Omron CX-Programmer project 新工程 (CX-Programmer 9.73)

# PLC 新PLC1: CQM1H CPU21

## Program 新程序1 (no task)
; 上传一个欧姆龙程序，轴承数控磨床用的。该程序控制三台步进电机。 / 系统涉及的物理设备包括操作面板按钮、传感器、砂轮电机、进给电机和冷却泵。 / 系统通过自动模式启动按钮启动整个流程，操作员按下后，工件在进给电机控制信号驱动下被送入加工位置，由工件位置传感器1确认到位后，砂轮电机控制信号激活砂轮开始磨削。 / 为确保加工质量，加工进行中标志置位时，冷却泵启动信号必须保持激活，提供持续的冷却液，防止工件过热损坏。 / 在加工进行中标志激活时，通过定时器确保冷却泵启动信号持续运行。 / 当工件位置传感器1确认工件到位后，砂轮电机控制信号才会被激活，避免空转浪费能源或损伤设备。 / 在手动模式下，进给电机启动按钮置位控制信号，进而驱动进给电机。 / 在自动模式启动按钮置位时，进给电机控制信号不会被手动触发。 / 进给过程中，进给脉冲信号根据数据存储区1设置的脉冲数精确控制步进电机，确保工件定位无偏差。 / 加工完成后，退料启用标志置位时，系统触发退料步骤将工件退出，避免工件滞留造成设备堵塞。 / 当退料启用标志置位时，若系统处于自动流程，触发退料步骤。 / 当工件位置传感器2检测工件离开时，流程结束并记录状态至数据存储区2。

### Section 段1

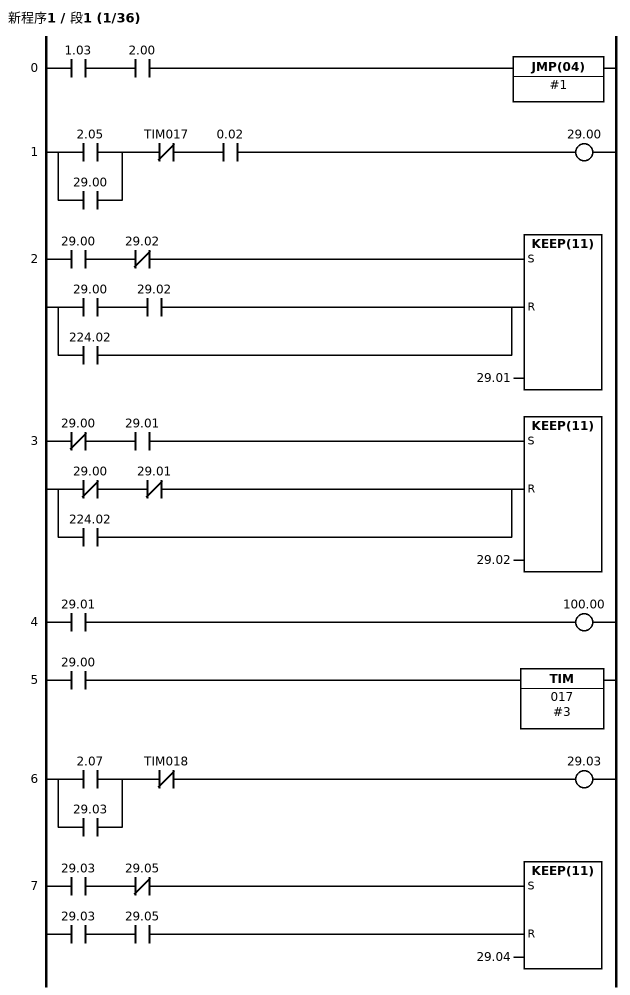
; rung 0
LD 1.03
AND 2.00
JMP(04) #1
; rung 1
LD 2.05
OR 29.00
ANDNOT TIM017
AND 0.02
OUT 29.00
; rung 2
LD 29.00
ANDNOT 29.02
LD 29.00
AND 29.02
OR 224.02
KEEP(11) 29.01
; rung 3
LDNOT 29.00
AND 29.01
LDNOT 29.00
ANDNOT 29.01
OR 224.02
KEEP(11) 29.02
; rung 4
LD 29.01
OUT 100.00
; rung 5
LD 29.00
TIM 017 #3
; rung 6
LD 2.07
OR 29.03
ANDNOT TIM018
OUT 29.03
; rung 7
LD 29.03
ANDNOT 29.05
LD 29.03
AND 29.05
KEEP(11) 29.04

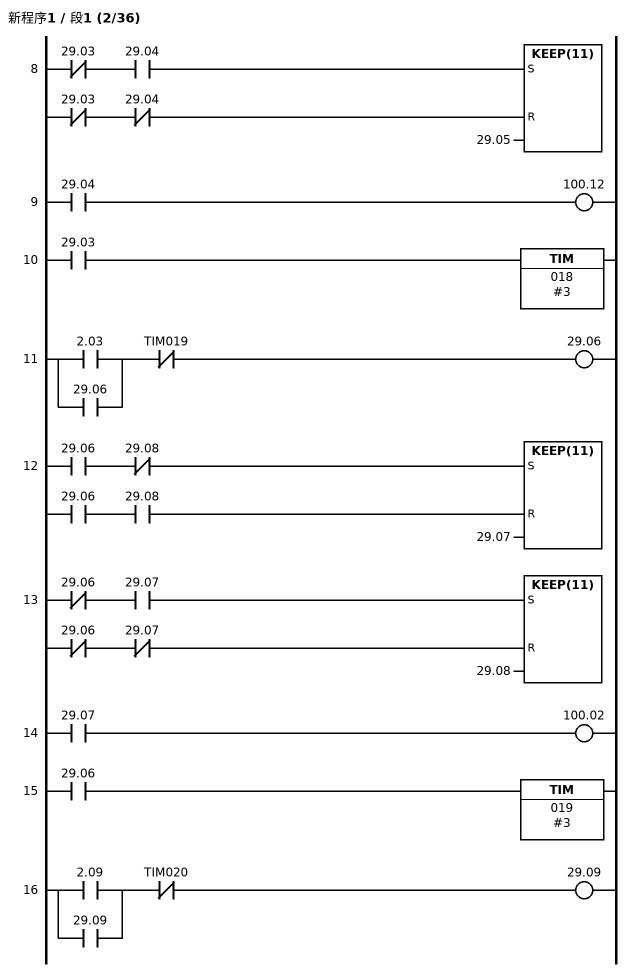
; rung 8
LDNOT 29.03
AND 29.04
LDNOT 29.03
ANDNOT 29.04
KEEP(11) 29.05
; rung 9
LD 29.04
OUT 100.12
; rung 10
LD 29.03
TIM 018 #3
; rung 11
LD 2.03
OR 29.06
ANDNOT TIM019
OUT 29.06
; rung 12
LD 29.06
ANDNOT 29.08
LD 29.06
AND 29.08
KEEP(11) 29.07
; rung 13
LDNOT 29.06
AND 29.07
LDNOT 29.06
ANDNOT 29.07
KEEP(11) 29.08
; rung 14
LD 29.07
OUT 100.02
; rung 15
LD 29.06
TIM 019 #3
; rung 16
LD 2.09
OR 29.09
ANDNOT TIM020
OUT 29.09

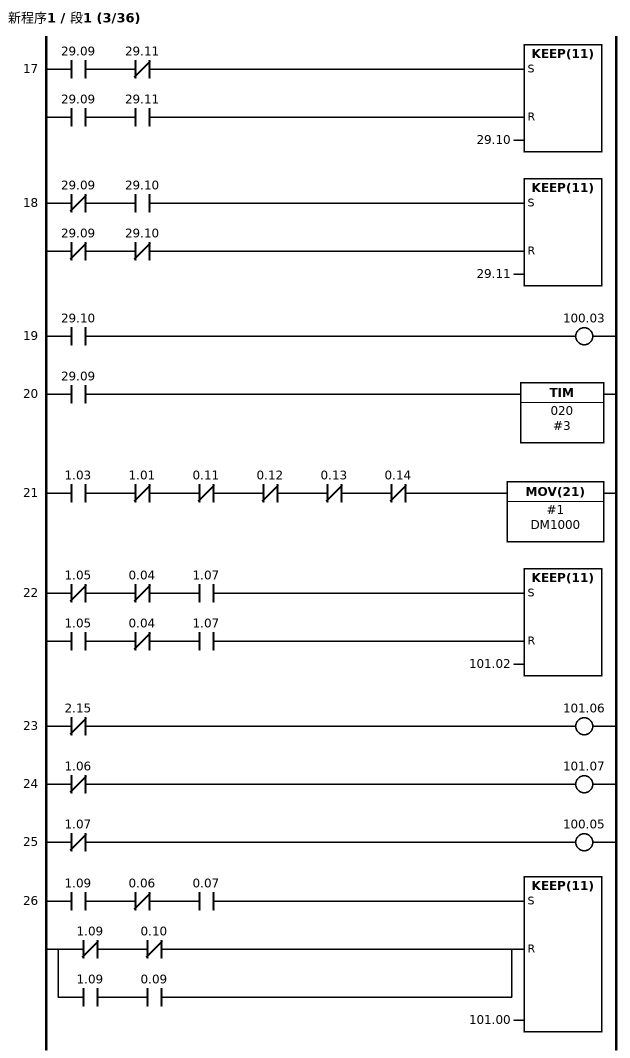
; rung 17
LD 29.09
ANDNOT 29.11
LD 29.09
AND 29.11
KEEP(11) 29.10
; rung 18
LDNOT 29.09
AND 29.10
LDNOT 29.09
ANDNOT 29.10
KEEP(11) 29.11
; rung 19
LD 29.10
OUT 100.03
; rung 20
LD 29.09
TIM 020 #3
; rung 21
LD 1.03
ANDNOT 1.01
ANDNOT 0.11
ANDNOT 0.12
ANDNOT 0.13
ANDNOT 0.14
MOV(21) #1 DM1000
; rung 22
LDNOT 1.05
ANDNOT 0.04
AND 1.07
LD 1.05
ANDNOT 0.04
AND 1.07
KEEP(11) 101.02
; rung 23
LDNOT 2.15
OUT 101.06
; rung 24
LDNOT 1.06
OUT 101.07
; rung 25
LDNOT 1.07
OUT 100.05
; rung 26
LD 1.09
ANDNOT 0.06
AND 0.07
LDNOT 1.09
ANDNOT 0.10
LD 1.09
AND 0.09
ORLD
KEEP(11) 101.00

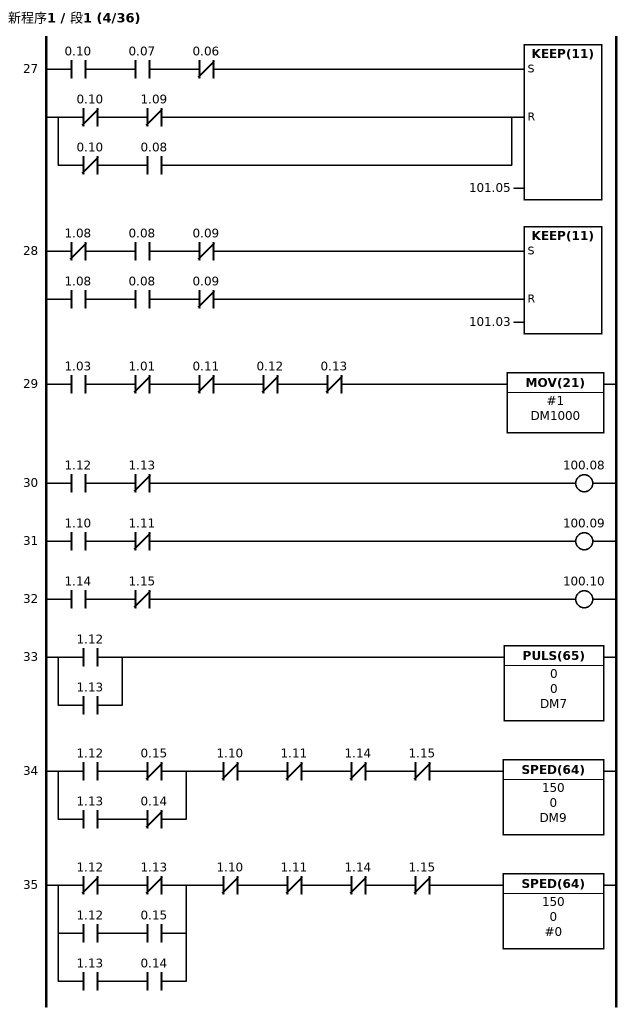
; rung 27
LD 0.10
AND 0.07
ANDNOT 0.06
LDNOT 0.10
ANDNOT 1.09
LDNOT 0.10
AND 0.08
ORLD
KEEP(11) 101.05
; rung 28
LDNOT 1.08
AND 0.08
ANDNOT 0.09
LD 1.08
AND 0.08
ANDNOT 0.09
KEEP(11) 101.03
; rung 29
LD 1.03
ANDNOT 1.01
ANDNOT 0.11
ANDNOT 0.12
ANDNOT 0.13
MOV(21) #1 DM1000
; rung 30
LD 1.12
ANDNOT 1.13
OUT 100.08
; rung 31
LD 1.10
ANDNOT 1.11
OUT 100.09
; rung 32
LD 1.14
ANDNOT 1.15
OUT 100.10
; rung 33
LD 1.12
OR 1.13
PULS(65) 0 0 DM7
; rung 34
LD 1.12
ANDNOT 0.15
LD 1.13
ANDNOT 0.14
ORLD
ANDNOT 1.10
ANDNOT 1.11
ANDNOT 1.14
ANDNOT 1.15
SPED(64) 150 0 DM9
; rung 35
LDNOT 1.12
ANDNOT 1.13
LD 1.12
AND 0.15
ORLD
LD 1.13
AND 0.14
ORLD
ANDNOT 1.10
ANDNOT 1.11
ANDNOT 1.14
ANDNOT 1.15
SPED(64) 150 0 #0

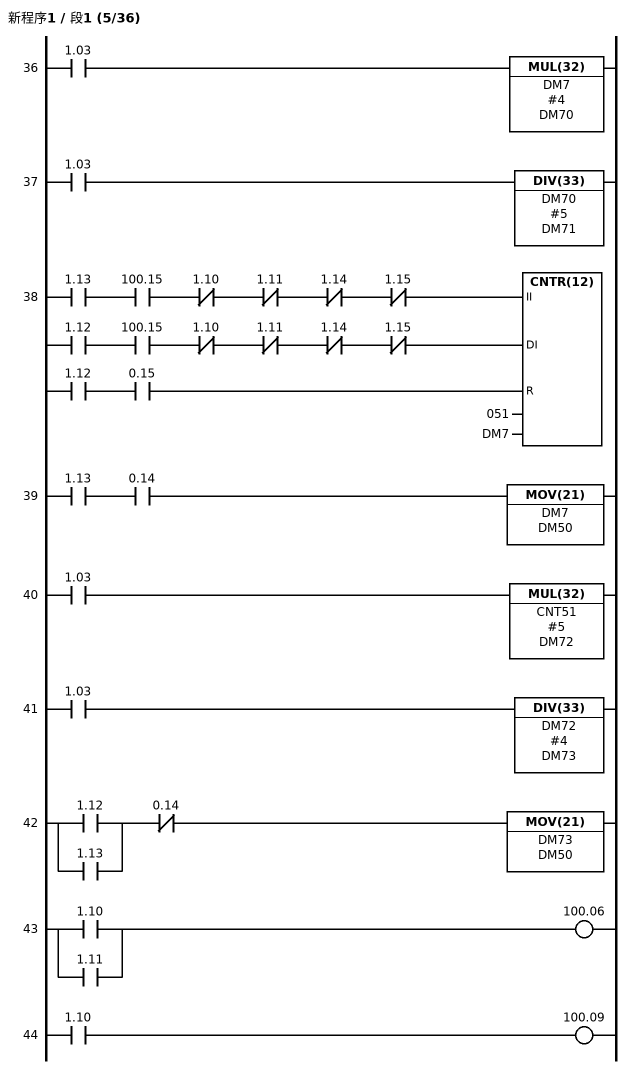
; rung 36
LD 1.03
MUL(32) DM7 #4 DM70
; rung 37
LD 1.03
DIV(33) DM70 #5 DM71
; rung 38
LD 1.13
AND 100.15
ANDNOT 1.10
ANDNOT 1.11
ANDNOT 1.14
ANDNOT 1.15
LD 1.12
AND 100.15
ANDNOT 1.10
ANDNOT 1.11
ANDNOT 1.14
ANDNOT 1.15
LD 1.12
AND 0.15
CNTR(12) 051 DM7
; rung 39
LD 1.13
AND 0.14
MOV(21) DM7 DM50
; rung 40
LD 1.03
MUL(32) CNT51 #5 DM72
; rung 41
LD 1.03
DIV(33) DM72 #4 DM73
; rung 42
LD 1.12
OR 1.13
ANDNOT 0.14
MOV(21) DM73 DM50
; rung 43
LD 1.10
OR 1.11
OUT 100.06
; rung 44
LD 1.10
OUT 100.09

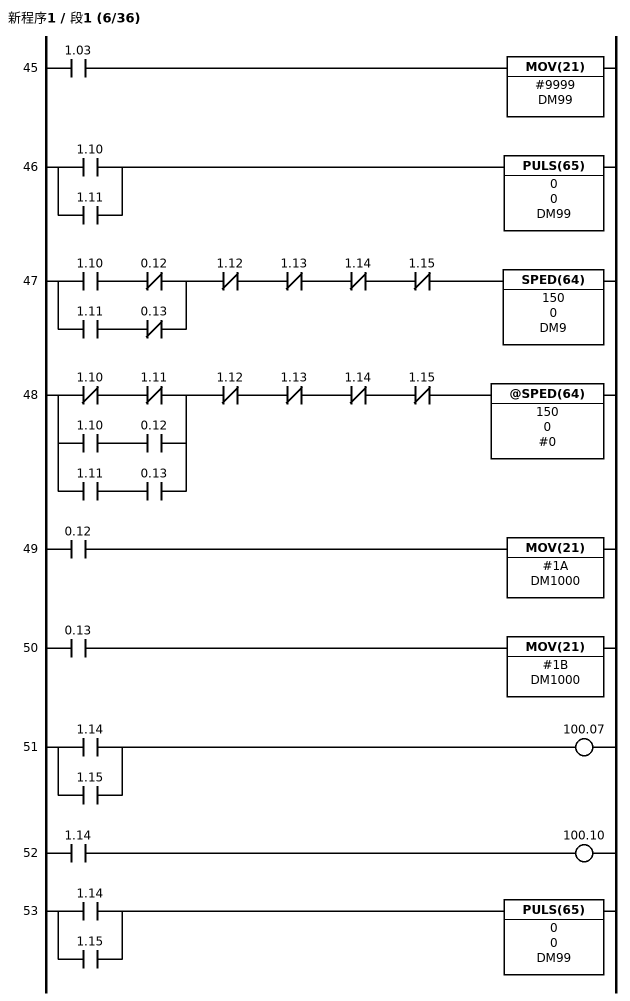
; rung 45
LD 1.03
MOV(21) #9999 DM99
; rung 46
LD 1.10
OR 1.11
PULS(65) 0 0 DM99
; rung 47
LD 1.10
ANDNOT 0.12
LD 1.11
ANDNOT 0.13
ORLD
ANDNOT 1.12
ANDNOT 1.13
ANDNOT 1.14
ANDNOT 1.15
SPED(64) 150 0 DM9
; rung 48
LDNOT 1.10
ANDNOT 1.11
LD 1.10
AND 0.12
ORLD
LD 1.11
AND 0.13
ORLD
ANDNOT 1.12
ANDNOT 1.13
ANDNOT 1.14
ANDNOT 1.15
@SPED(64) 150 0 #0
; rung 49
LD 0.12
MOV(21) #1A DM1000
; rung 50
LD 0.13
MOV(21) #1B DM1000
; rung 51
LD 1.14
OR 1.15
OUT 100.07
; rung 52
LD 1.14
OUT 100.10
; rung 53
LD 1.14
OR 1.15
PULS(65) 0 0 DM99

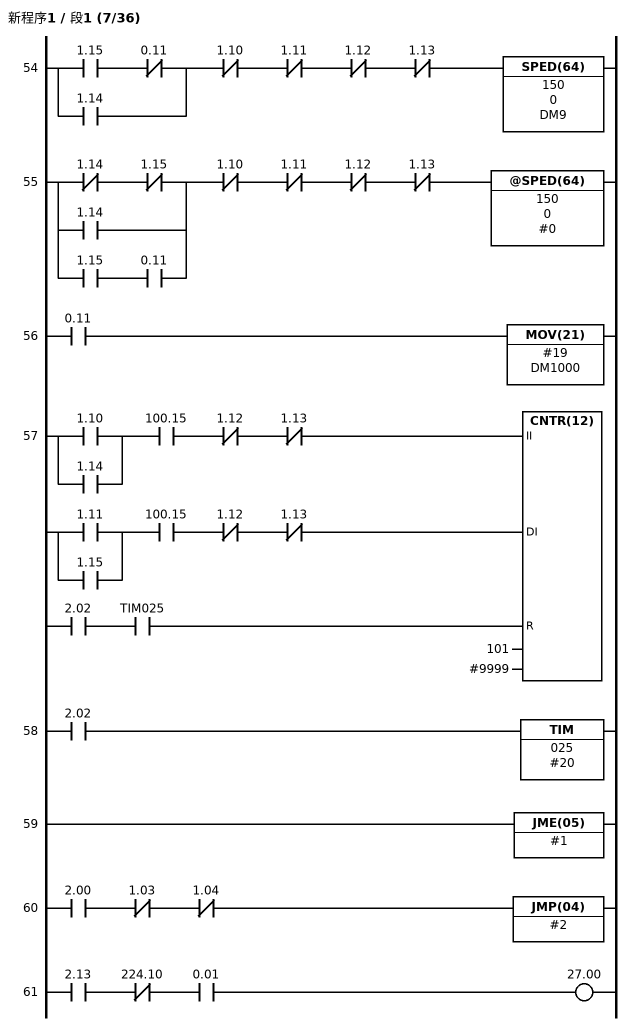
; rung 54
LD 1.15
ANDNOT 0.11
OR 1.14
ANDNOT 1.10
ANDNOT 1.11
ANDNOT 1.12
ANDNOT 1.13
SPED(64) 150 0 DM9
; rung 55
LDNOT 1.14
ANDNOT 1.15
OR 1.14
LD 1.15
AND 0.11
ORLD
ANDNOT 1.10
ANDNOT 1.11
ANDNOT 1.12
ANDNOT 1.13
@SPED(64) 150 0 #0
; rung 56
LD 0.11
MOV(21) #19 DM1000
; rung 57
LD 1.10
OR 1.14
AND 100.15
ANDNOT 1.12
ANDNOT 1.13
LD 1.11
OR 1.15
AND 100.15
ANDNOT 1.12
ANDNOT 1.13
LD 2.02
AND TIM025
CNTR(12) 101 #9999
; rung 58
LD 2.02
TIM 025 #20
; rung 59
JME(05) #1
; rung 60
LD 2.00
ANDNOT 1.03
ANDNOT 1.04
JMP(04) #2
; rung 61
LD 2.13
ANDNOT 224.10
AND 0.01
OUT 27.00

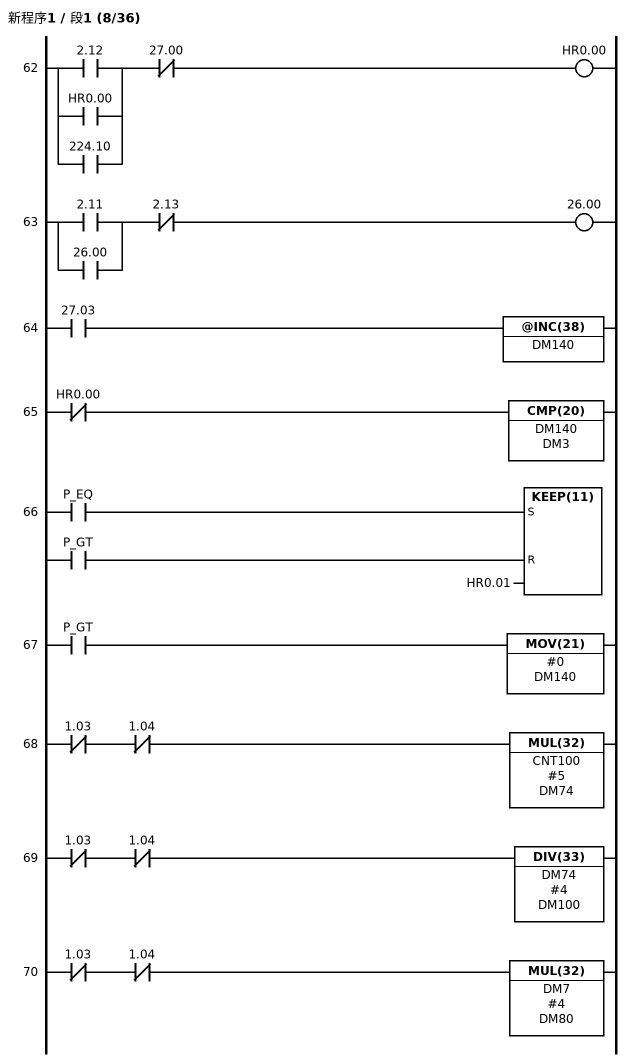
; rung 62
LD 2.12
OR HR0.00
OR 224.10
ANDNOT 27.00
OUT HR0.00
; rung 63
LD 2.11
OR 26.00
ANDNOT 2.13
OUT 26.00
; rung 64
LD 27.03
@INC(38) DM140
; rung 65
LDNOT HR0.00
CMP(20) DM140 DM3
; rung 66
LD P_EQ
LD P_GT
KEEP(11) HR0.01
; rung 67
LD P_GT
MOV(21) #0 DM140
; rung 68
LDNOT 1.03
ANDNOT 1.04
MUL(32) CNT100 #5 DM74
; rung 69
LDNOT 1.03
ANDNOT 1.04
DIV(33) DM74 #4 DM100
; rung 70
LDNOT 1.03
ANDNOT 1.04
MUL(32) DM7 #4 DM80

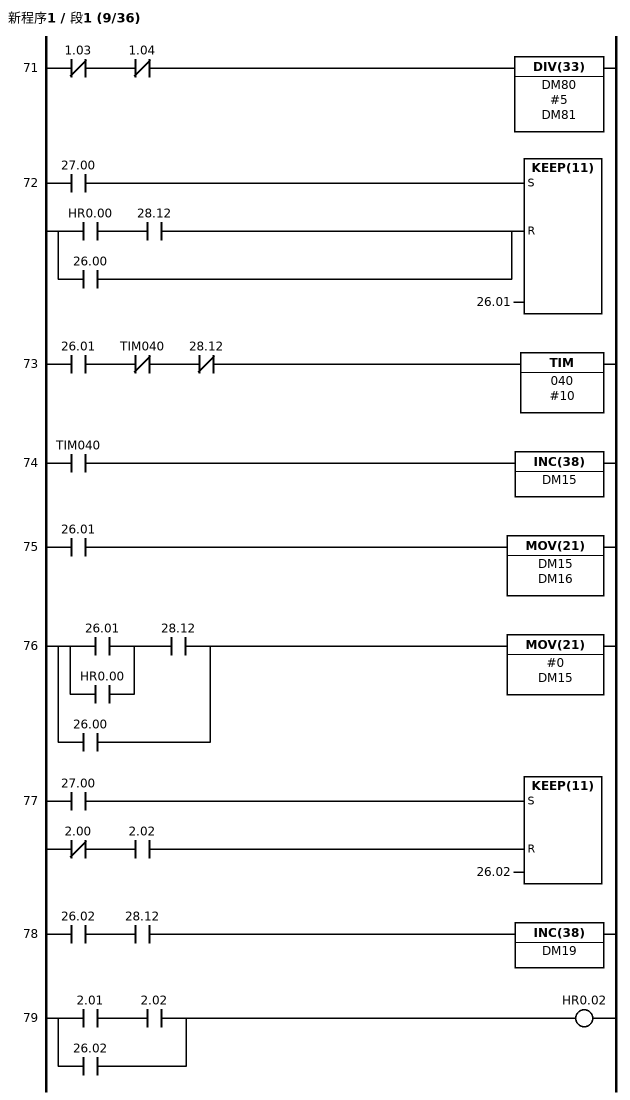
; rung 71
LDNOT 1.03
ANDNOT 1.04
DIV(33) DM80 #5 DM81
; rung 72
LD 27.00
LD HR0.00
AND 28.12
OR 26.00
KEEP(11) 26.01
; rung 73
LD 26.01
ANDNOT TIM040
ANDNOT 28.12
TIM 040 #10
; rung 74
LD TIM040
INC(38) DM15
; rung 75
LD 26.01
MOV(21) DM15 DM16
; rung 76
LD 26.01
OR HR0.00
AND 28.12
OR 26.00
MOV(21) #0 DM15
; rung 77
LD 27.00
LDNOT 2.00
AND 2.02
KEEP(11) 26.02
; rung 78
LD 26.02
AND 28.12
INC(38) DM19
; rung 79
LD 2.01
AND 2.02
OR 26.02
OUT HR0.02

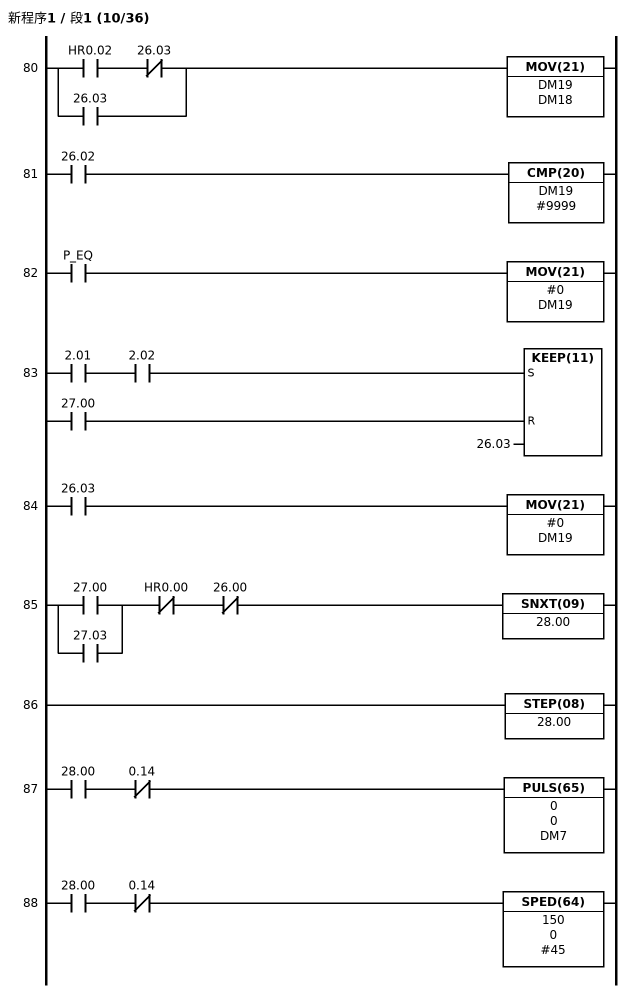
; rung 80
LD HR0.02
ANDNOT 26.03
OR 26.03
MOV(21) DM19 DM18
; rung 81
LD 26.02
CMP(20) DM19 #9999
; rung 82
LD P_EQ
MOV(21) #0 DM19
; rung 83
LD 2.01
AND 2.02
LD 27.00
KEEP(11) 26.03
; rung 84
LD 26.03
MOV(21) #0 DM19
; rung 85
LD 27.00
OR 27.03
ANDNOT HR0.00
ANDNOT 26.00
SNXT(09) 28.00
; rung 86
STEP(08) 28.00
; rung 87
LD 28.00
ANDNOT 0.14
PULS(65) 0 0 DM7
; rung 88
LD 28.00
ANDNOT 0.14
SPED(64) 150 0 #45

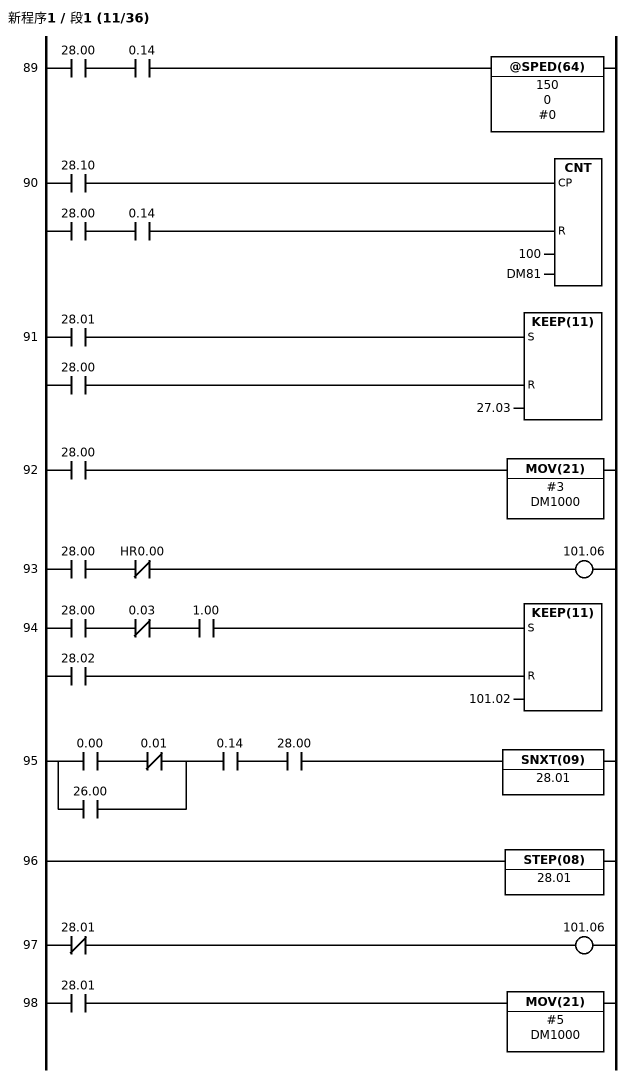
; rung 89
LD 28.00
AND 0.14
@SPED(64) 150 0 #0
; rung 90
LD 28.10
LD 28.00
AND 0.14
CNT 100 DM81
; rung 91
LD 28.01
LD 28.00
KEEP(11) 27.03
; rung 92
LD 28.00
MOV(21) #3 DM1000
; rung 93
LD 28.00
ANDNOT HR0.00
OUT 101.06
; rung 94
LD 28.00
ANDNOT 0.03
AND 1.00
LD 28.02
KEEP(11) 101.02
; rung 95
LD 0.00
ANDNOT 0.01
OR 26.00
AND 0.14
AND 28.00
SNXT(09) 28.01
; rung 96
STEP(08) 28.01
; rung 97
LDNOT 28.01
OUT 101.06
; rung 98
LD 28.01
MOV(21) #5 DM1000

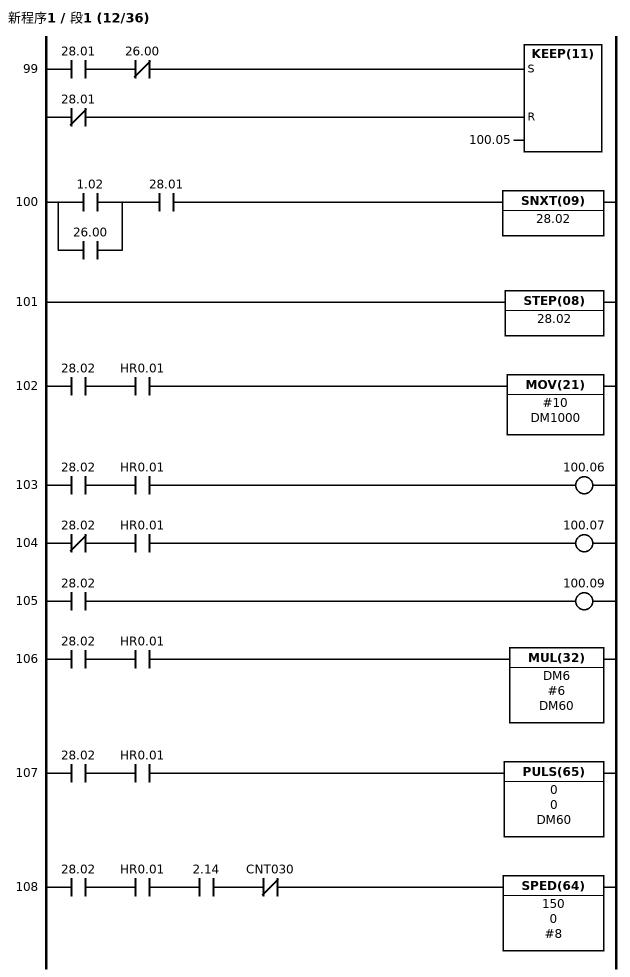
; rung 99
LD 28.01
ANDNOT 26.00
LDNOT 28.01
KEEP(11) 100.05
; rung 100
LD 1.02
OR 26.00
AND 28.01
SNXT(09) 28.02
; rung 101
STEP(08) 28.02
; rung 102
LD 28.02
AND HR0.01
MOV(21) #10 DM1000
; rung 103
LD 28.02
AND HR0.01
OUT 100.06
; rung 104
LDNOT 28.02
AND HR0.01
OUT 100.07
; rung 105
LD 28.02
OUT 100.09
; rung 106
LD 28.02
AND HR0.01
MUL(32) DM6 #6 DM60
; rung 107
LD 28.02
AND HR0.01
PULS(65) 0 0 DM60
; rung 108
LD 28.02
AND HR0.01
AND 2.14
ANDNOT CNT030
SPED(64) 150 0 #8

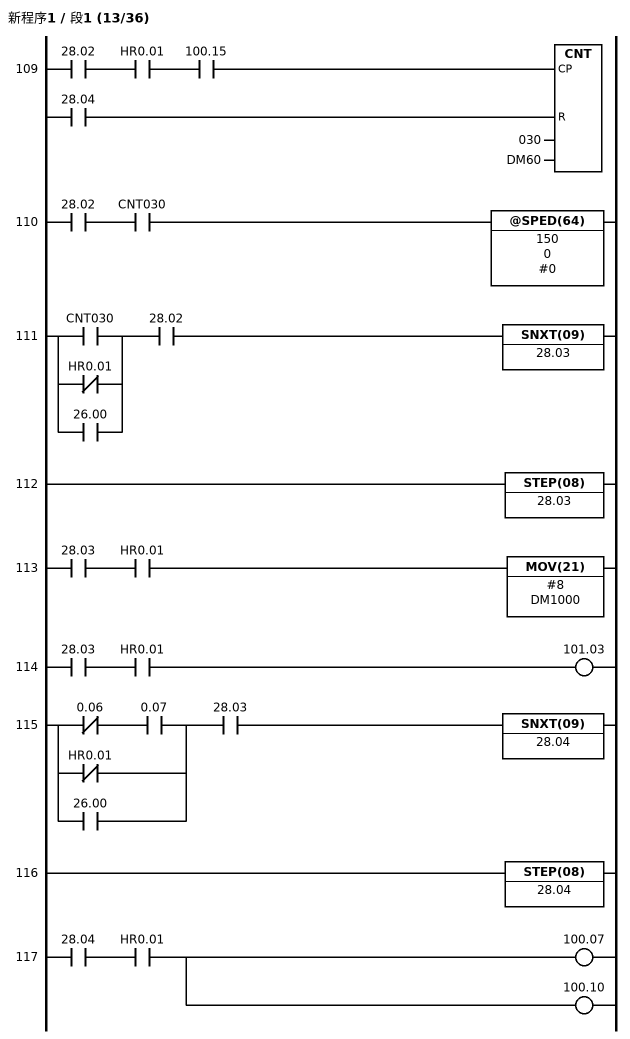
; rung 109
LD 28.02
AND HR0.01
AND 100.15
LD 28.04
CNT 030 DM60
; rung 110
LD 28.02
AND CNT030
@SPED(64) 150 0 #0
; rung 111
LD CNT030
ORNOT HR0.01
OR 26.00
AND 28.02
SNXT(09) 28.03
; rung 112
STEP(08) 28.03
; rung 113
LD 28.03
AND HR0.01
MOV(21) #8 DM1000
; rung 114
LD 28.03
AND HR0.01
OUT 101.03
; rung 115
LDNOT 0.06
AND 0.07
ORNOT HR0.01
OR 26.00
AND 28.03
SNXT(09) 28.04
; rung 116
STEP(08) 28.04
; rung 117
LD 28.04
AND HR0.01
OUT 100.07
OUT 100.10

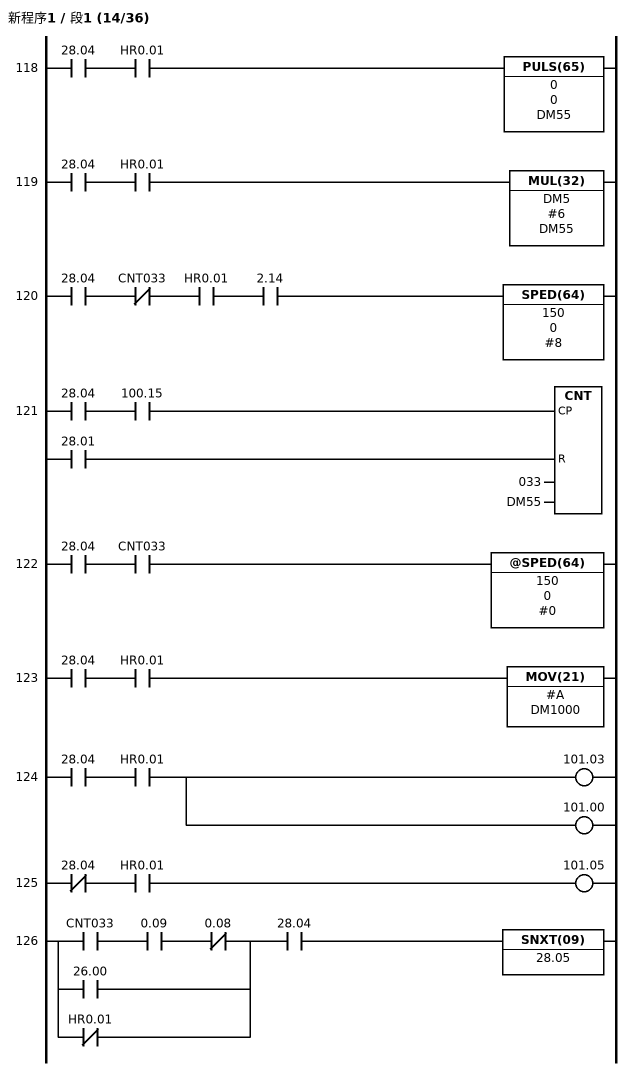
; rung 118
LD 28.04
AND HR0.01
PULS(65) 0 0 DM55
; rung 119
LD 28.04
AND HR0.01
MUL(32) DM5 #6 DM55
; rung 120
LD 28.04
ANDNOT CNT033
AND HR0.01
AND 2.14
SPED(64) 150 0 #8
; rung 121
LD 28.04
AND 100.15
LD 28.01
CNT 033 DM55
; rung 122
LD 28.04
AND CNT033
@SPED(64) 150 0 #0
; rung 123
LD 28.04
AND HR0.01
MOV(21) #A DM1000
; rung 124
LD 28.04
AND HR0.01
OUT 101.03
OUT 101.00
; rung 125
LDNOT 28.04
AND HR0.01
OUT 101.05
; rung 126
LD CNT033
AND 0.09
ANDNOT 0.08
OR 26.00
ORNOT HR0.01
AND 28.04
SNXT(09) 28.05

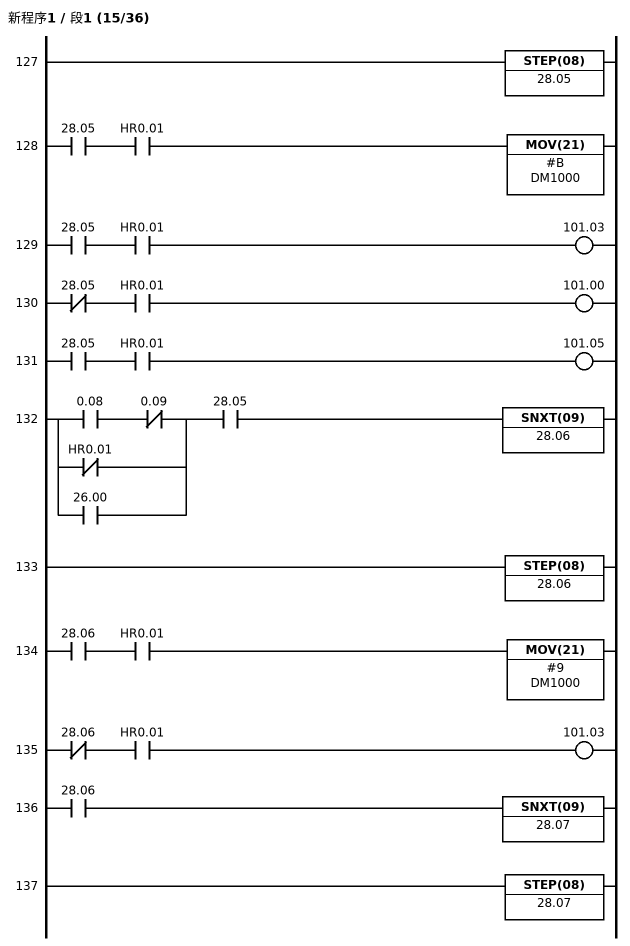
; rung 127
STEP(08) 28.05
; rung 128
LD 28.05
AND HR0.01
MOV(21) #B DM1000
; rung 129
LD 28.05
AND HR0.01
OUT 101.03
; rung 130
LDNOT 28.05
AND HR0.01
OUT 101.00
; rung 131
LD 28.05
AND HR0.01
OUT 101.05
; rung 132
LD 0.08
ANDNOT 0.09
ORNOT HR0.01
OR 26.00
AND 28.05
SNXT(09) 28.06
; rung 133
STEP(08) 28.06
; rung 134
LD 28.06
AND HR0.01
MOV(21) #9 DM1000
; rung 135
LDNOT 28.06
AND HR0.01
OUT 101.03
; rung 136
LD 28.06
SNXT(09) 28.07
; rung 137
STEP(08) 28.07

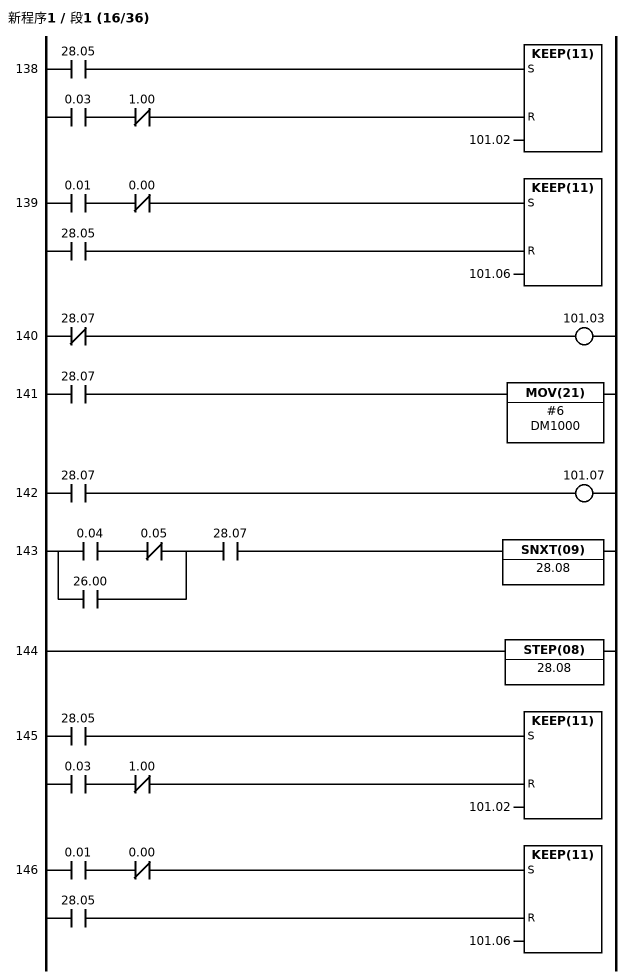
; rung 138
LD 28.05
LD 0.03
ANDNOT 1.00
KEEP(11) 101.02
; rung 139
LD 0.01
ANDNOT 0.00
LD 28.05
KEEP(11) 101.06
; rung 140
LDNOT 28.07
OUT 101.03
; rung 141
LD 28.07
MOV(21) #6 DM1000
; rung 142
LD 28.07
OUT 101.07
; rung 143
LD 0.04
ANDNOT 0.05
OR 26.00
AND 28.07
SNXT(09) 28.08
; rung 144
STEP(08) 28.08
; rung 145
LD 28.05
LD 0.03
ANDNOT 1.00
KEEP(11) 101.02
; rung 146
LD 0.01
ANDNOT 0.00
LD 28.05
KEEP(11) 101.06

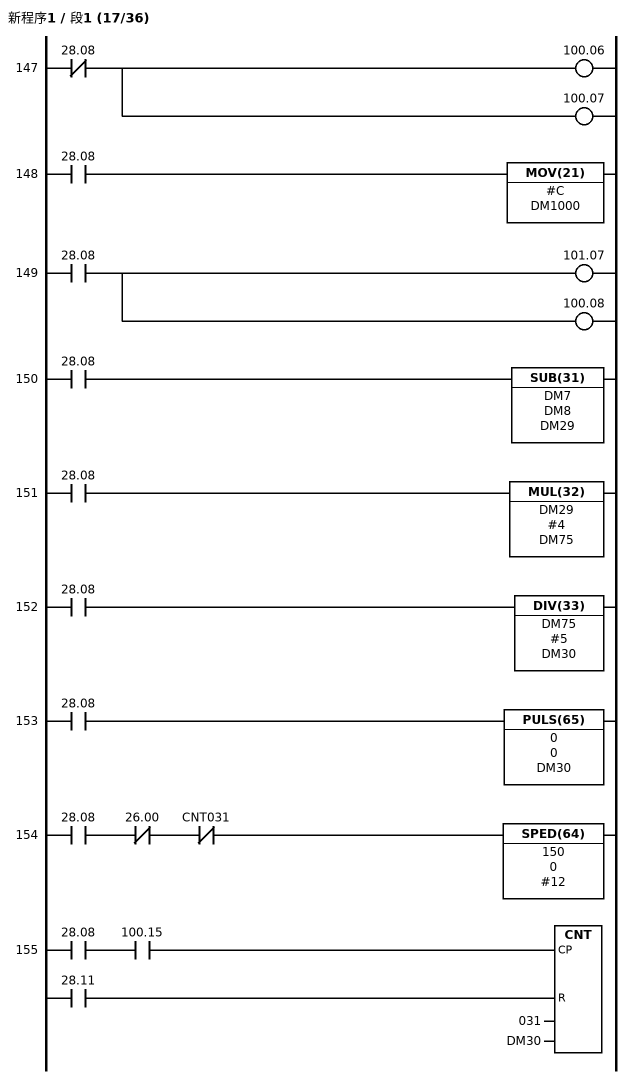
; rung 147
LDNOT 28.08
OUT 100.06
OUT 100.07
; rung 148
LD 28.08
MOV(21) #C DM1000
; rung 149
LD 28.08
OUT 101.07
OUT 100.08
; rung 150
LD 28.08
SUB(31) DM7 DM8 DM29
; rung 151
LD 28.08
MUL(32) DM29 #4 DM75
; rung 152
LD 28.08
DIV(33) DM75 #5 DM30
; rung 153
LD 28.08
PULS(65) 0 0 DM30
; rung 154
LD 28.08
ANDNOT 26.00
ANDNOT CNT031
SPED(64) 150 0 #12
; rung 155
LD 28.08
AND 100.15
LD 28.11
CNT 031 DM30

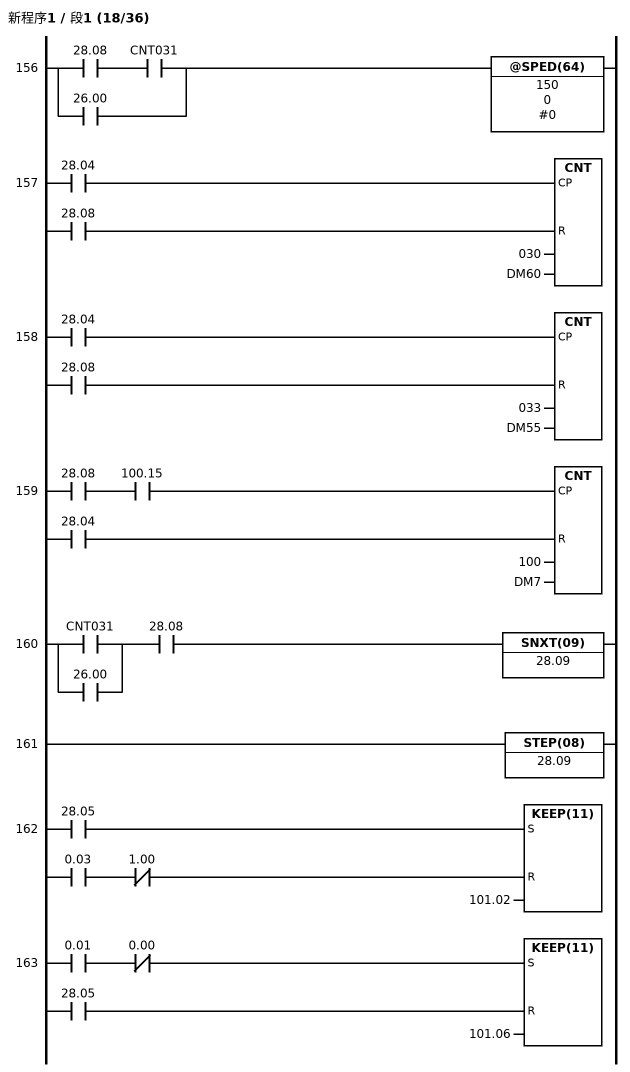
; rung 156
LD 28.08
AND CNT031
OR 26.00
@SPED(64) 150 0 #0
; rung 157
LD 28.04
LD 28.08
CNT 030 DM60
; rung 158
LD 28.04
LD 28.08
CNT 033 DM55
; rung 159
LD 28.08
AND 100.15
LD 28.04
CNT 100 DM7
; rung 160
LD CNT031
OR 26.00
AND 28.08
SNXT(09) 28.09
; rung 161
STEP(08) 28.09
; rung 162
LD 28.05
LD 0.03
ANDNOT 1.00
KEEP(11) 101.02
; rung 163
LD 0.01
ANDNOT 0.00
LD 28.05
KEEP(11) 101.06

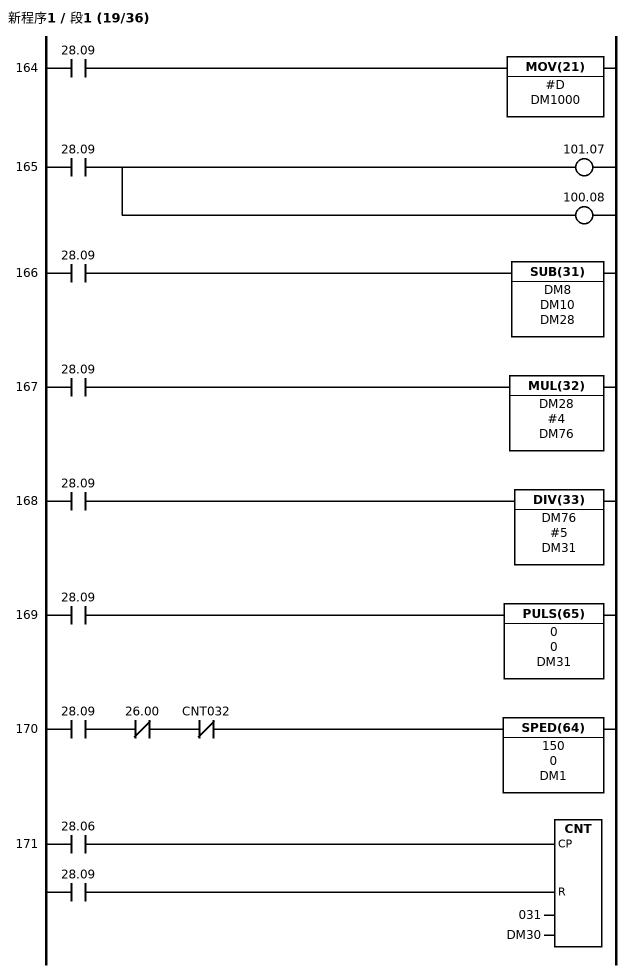
; rung 164
LD 28.09
MOV(21) #D DM1000
; rung 165
LD 28.09
OUT 101.07
OUT 100.08
; rung 166
LD 28.09
SUB(31) DM8 DM10 DM28
; rung 167
LD 28.09
MUL(32) DM28 #4 DM76
; rung 168
LD 28.09
DIV(33) DM76 #5 DM31
; rung 169
LD 28.09
PULS(65) 0 0 DM31
; rung 170
LD 28.09
ANDNOT 26.00
ANDNOT CNT032
SPED(64) 150 0 DM1
; rung 171
LD 28.06
LD 28.09
CNT 031 DM30

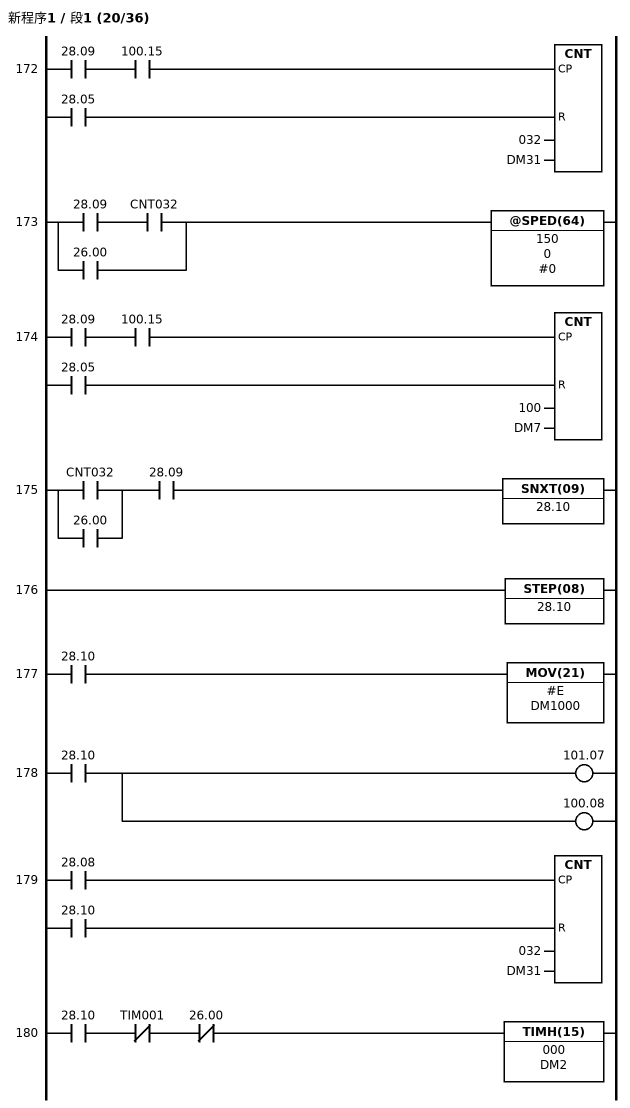
; rung 172
LD 28.09
AND 100.15
LD 28.05
CNT 032 DM31
; rung 173
LD 28.09
AND CNT032
OR 26.00
@SPED(64) 150 0 #0
; rung 174
LD 28.09
AND 100.15
LD 28.05
CNT 100 DM7
; rung 175
LD CNT032
OR 26.00
AND 28.09
SNXT(09) 28.10
; rung 176
STEP(08) 28.10
; rung 177
LD 28.10
MOV(21) #E DM1000
; rung 178
LD 28.10
OUT 101.07
OUT 100.08
; rung 179
LD 28.08
LD 28.10
CNT 032 DM31
; rung 180
LD 28.10
ANDNOT TIM001
ANDNOT 26.00
TIMH(15) 000 DM2

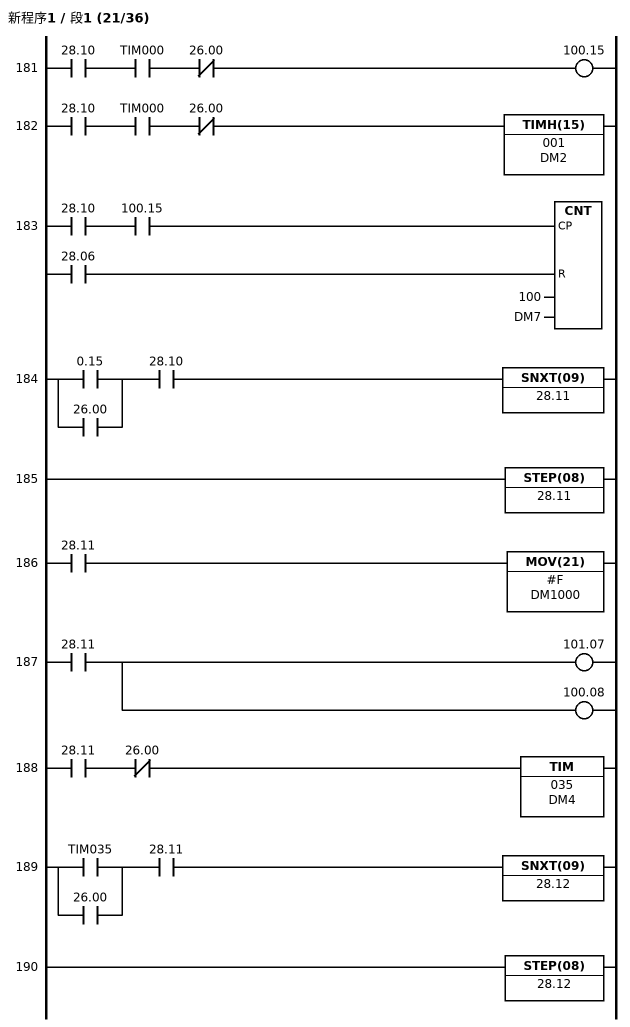
; rung 181
LD 28.10
AND TIM000
ANDNOT 26.00
OUT 100.15
; rung 182
LD 28.10
AND TIM000
ANDNOT 26.00
TIMH(15) 001 DM2
; rung 183
LD 28.10
AND 100.15
LD 28.06
CNT 100 DM7
; rung 184
LD 0.15
OR 26.00
AND 28.10
SNXT(09) 28.11
; rung 185
STEP(08) 28.11
; rung 186
LD 28.11
MOV(21) #F DM1000
; rung 187
LD 28.11
OUT 101.07
OUT 100.08
; rung 188
LD 28.11
ANDNOT 26.00
TIM 035 DM4
; rung 189
LD TIM035
OR 26.00
AND 28.11
SNXT(09) 28.12
; rung 190
STEP(08) 28.12

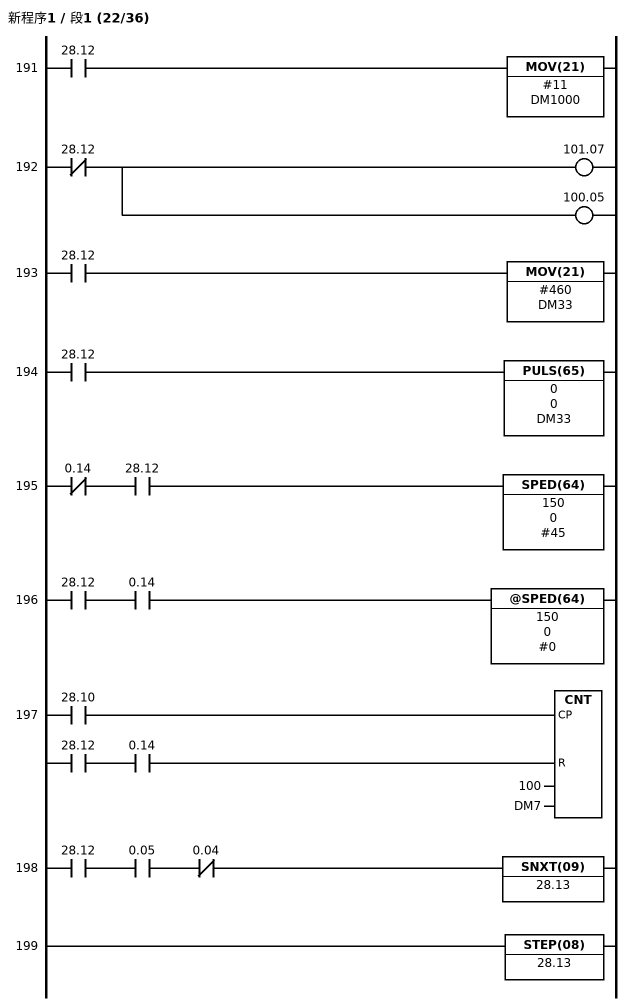
; rung 191
LD 28.12
MOV(21) #11 DM1000
; rung 192
LDNOT 28.12
OUT 101.07
OUT 100.05
; rung 193
LD 28.12
MOV(21) #460 DM33
; rung 194
LD 28.12
PULS(65) 0 0 DM33
; rung 195
LDNOT 0.14
AND 28.12
SPED(64) 150 0 #45
; rung 196
LD 28.12
AND 0.14
@SPED(64) 150 0 #0
; rung 197
LD 28.10
LD 28.12
AND 0.14
CNT 100 DM7
; rung 198
LD 28.12
AND 0.05
ANDNOT 0.04
SNXT(09) 28.13
; rung 199
STEP(08) 28.13

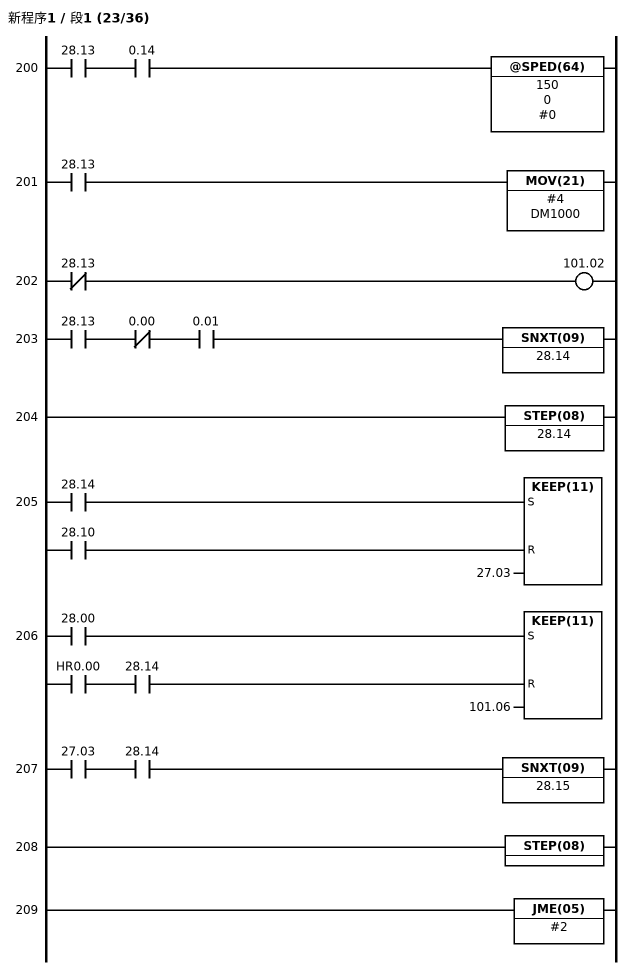
; rung 200
LD 28.13
AND 0.14
@SPED(64) 150 0 #0
; rung 201
LD 28.13
MOV(21) #4 DM1000
; rung 202
LDNOT 28.13
OUT 101.02
; rung 203
LD 28.13
ANDNOT 0.00
AND 0.01
SNXT(09) 28.14
; rung 204
STEP(08) 28.14
; rung 205
LD 28.14
LD 28.10
KEEP(11) 27.03
; rung 206
LD 28.00
LD HR0.00
AND 28.14
KEEP(11) 101.06
; rung 207
LD 27.03
AND 28.14
SNXT(09) 28.15
; rung 208
STEP(08)
; rung 209
JME(05) #2

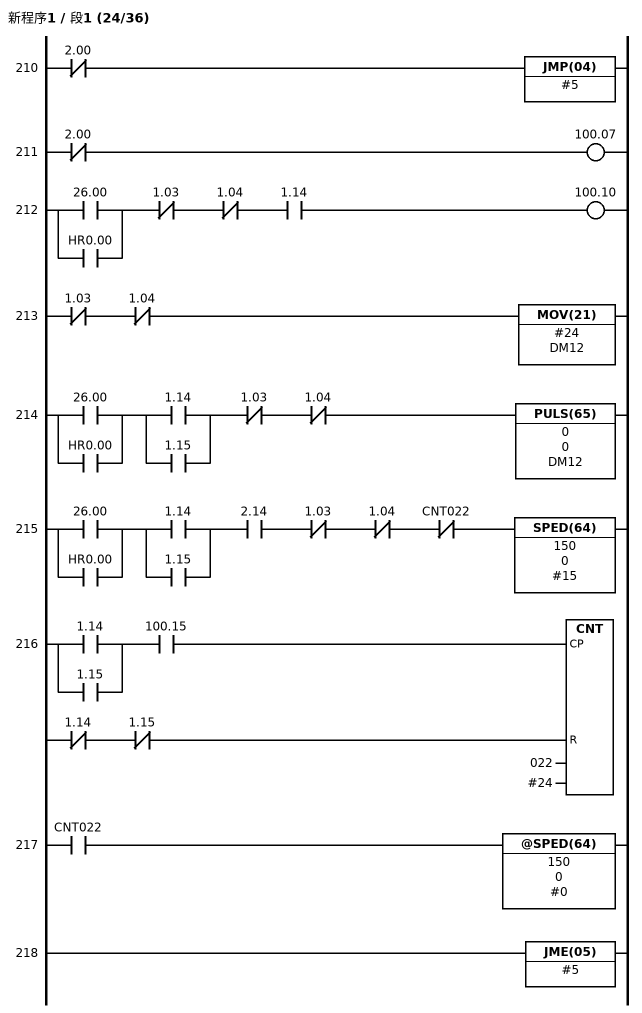
; rung 210
LDNOT 2.00
JMP(04) #5
; rung 211
LDNOT 2.00
OUT 100.07
; rung 212
LD 26.00
OR HR0.00
ANDNOT 1.03
ANDNOT 1.04
AND 1.14
OUT 100.10
; rung 213
LDNOT 1.03
ANDNOT 1.04
MOV(21) #24 DM12
; rung 214
LD 26.00
OR HR0.00
LD 1.14
OR 1.15
ANDLD
ANDNOT 1.03
ANDNOT 1.04
PULS(65) 0 0 DM12
; rung 215
LD 26.00
OR HR0.00
LD 1.14
OR 1.15
ANDLD
AND 2.14
ANDNOT 1.03
ANDNOT 1.04
ANDNOT CNT022
SPED(64) 150 0 #15
; rung 216
LD 1.14
OR 1.15
AND 100.15
LDNOT 1.14
ANDNOT 1.15
CNT 022 #24
; rung 217
LD CNT022
@SPED(64) 150 0 #0
; rung 218
JME(05) #5

